TYPE ST_LogMessage :
STRUCT
  iTyp : INT; // 0=hint 1=warning 2=error
  dtDateTime : DATE_AND_TIME;
  szPath : STRING(60);
  szMessage : STRING(80);
END_STRUCT
END_TYPE

(* stored: Version 1.1.0.1, ProductVersion 3.1.4018.9
   DUT ST_LogMessage: Id {259e617e-3a06-4b53-b74e-3e74400c9fee} *)
